// TwinCAT 3 PLC project SARUtils
// Title: SARUtills
// Company: Stian Arevoll
// Author: Stian Arevoll
// ProjectVersion: 0.1.2
// ProgramVersion: 3.1.4024.0
// libraries:
//   Tc2_System, * (Beckhoff Automation GmbH)
//   Tc2_Utilities, * (Beckhoff Automation GmbH)
//   Tc3_Module, * (Beckhoff Automation GmbH)
//   TcUnit, * (www.tcunit.org)
// project tree:
//   / PlcTask.TcTTO
//   POUs/ FB_Concater.TcPOU (not stored), I_Concater.TcIO (not stored)
//   Tests/ FB_Concater_Test.TcPOU (not stored), P_Concater_Tests.TcPOU

CONFIGURATION SARUtils
    RESOURCE PLC ON TwinCAT3
        TASK PlcTask(INTERVAL := T#10ms, PRIORITY := 20);
    END_RESOURCE
END_CONFIGURATION

// ---- Tests/P_Concater_Tests.TcPOU
PROGRAM P_Concater_Tests
VAR
	fbConcater_Test : FB_Concater_Test;
END_VAR

TcUnit.RUN();

END_PROGRAM
